// SIMATIC S7-200 project (STEP 7-Micro/WIN), CPU 224 CN REL 02.01

ORGANIZATION_BLOCK 主程序:OB1
TITLE=程序注释
BEGIN
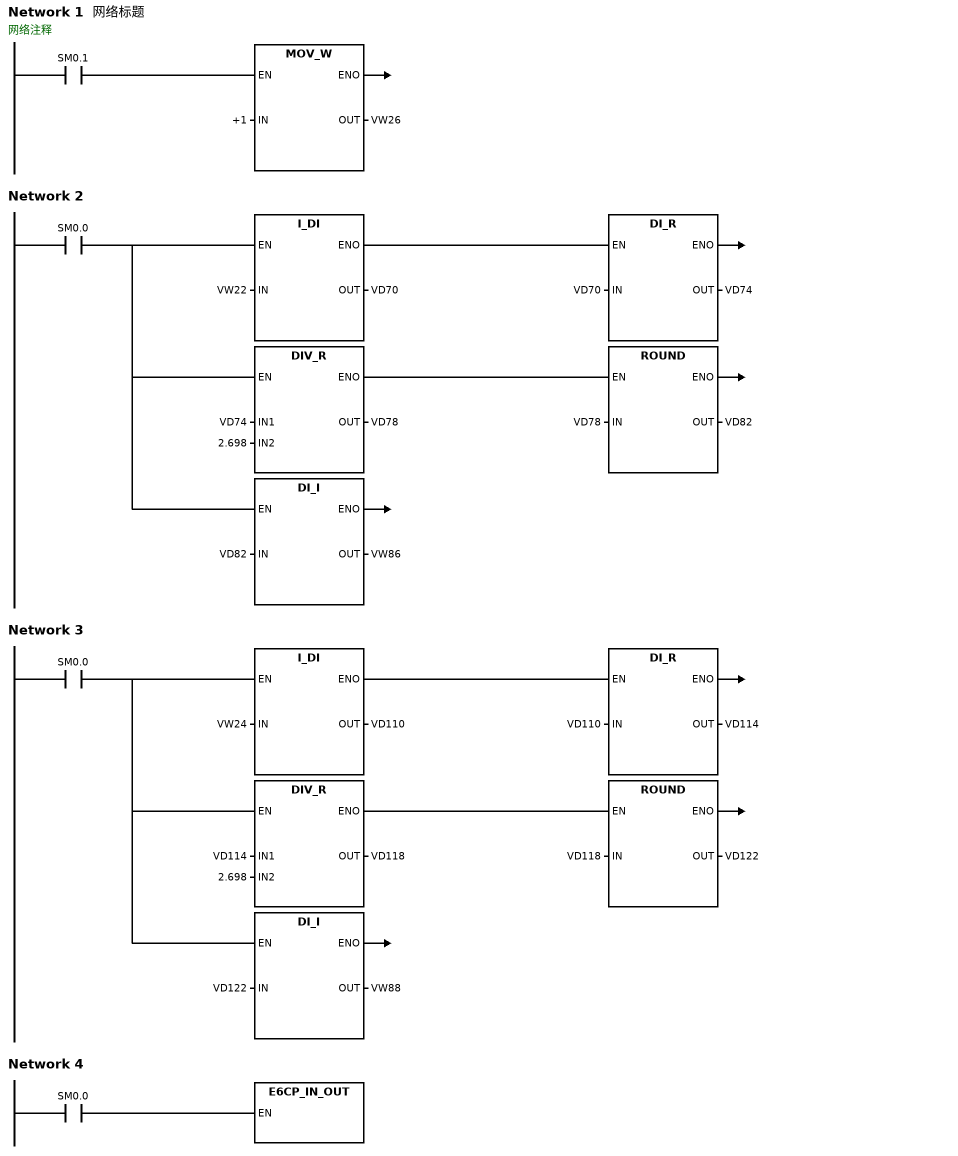
Network 1 // 网络标题
// 网络注释
LD     SM0.1
MOVW   +1, VW26
Network 2
LD     SM0.0
LPS
ITD    VW22, VD70
AENO
DTR    VD70, VD74
LRD
MOVR   VD74, VD78
AENO
/R     2.698, VD78
AENO
ROUND  VD78, VD82
LPP
DTI    VD82, VW86
Network 3
LD     SM0.0
LPS
ITD    VW24, VD110
AENO
DTR    VD110, VD114
LRD
MOVR   VD114, VD118
AENO
/R     2.698, VD118
AENO
ROUND  VD118, VD122
LPP
DTI    VD122, VW88
Network 4
LD     SM0.0
CALL   E6CP_IN_OUT:SBR4
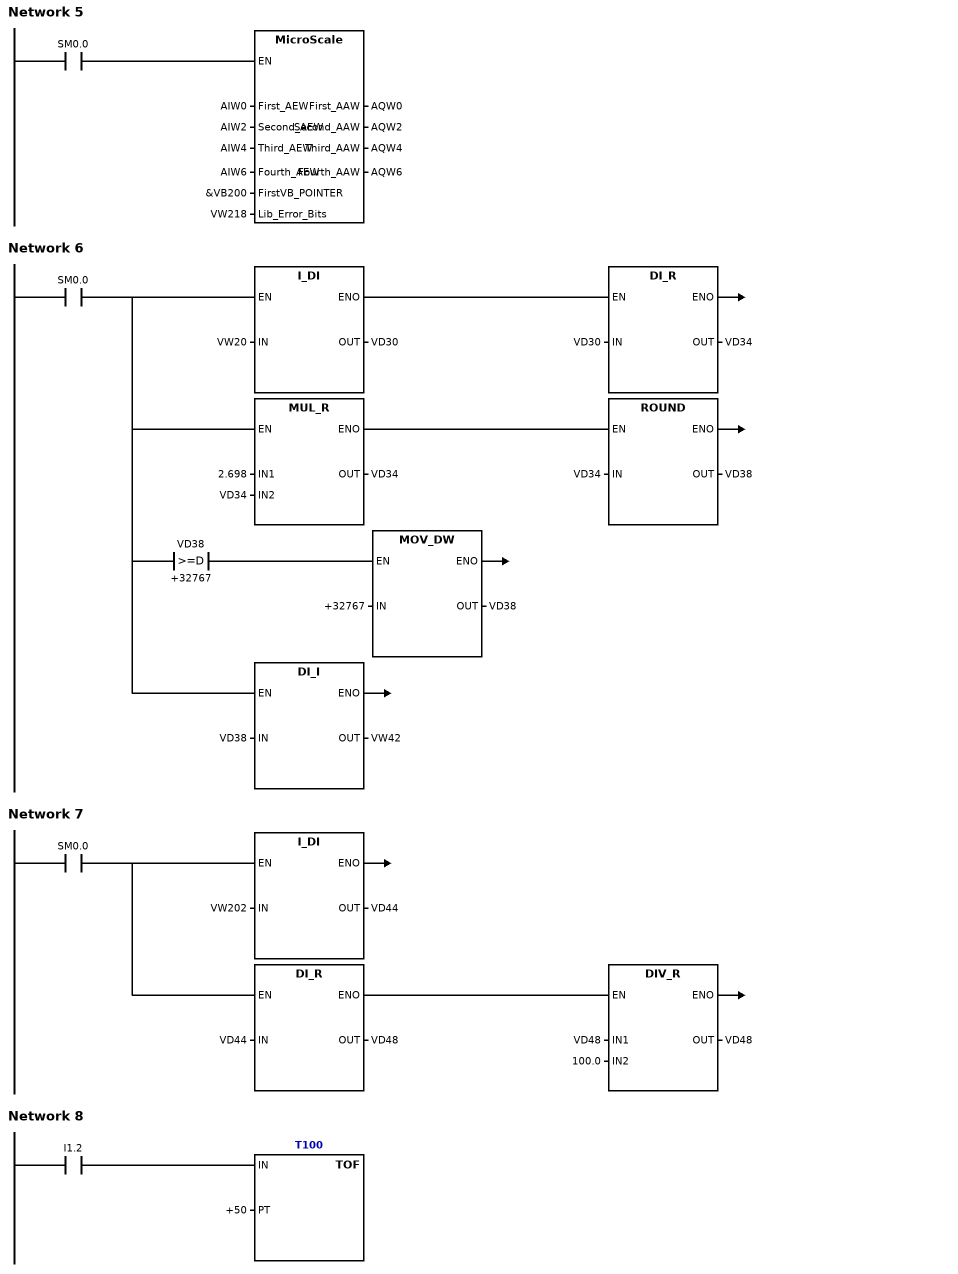
Network 5
LD     SM0.0
CALL   MicroScale:SBR3, AIW0, AIW2, AIW4, AIW6, &VB200, VW218, AQW0, AQW2, AQW4, AQW6
Network 6
LD     SM0.0
LPS
ITD    VW20, VD30
AENO
DTR    VD30, VD34
LRD
*R     2.698, VD34
AENO
ROUND  VD34, VD38
LRD
AD>=   VD38, +32767
MOVD   +32767, VD38
LPP
DTI    VD38, VW42
Network 7
LD     SM0.0
ITD    VW202, VD44
DTR    VD44, VD48
AENO
/R     100.0, VD48
Network 8
LD     I1.2
TOF    T100, +50
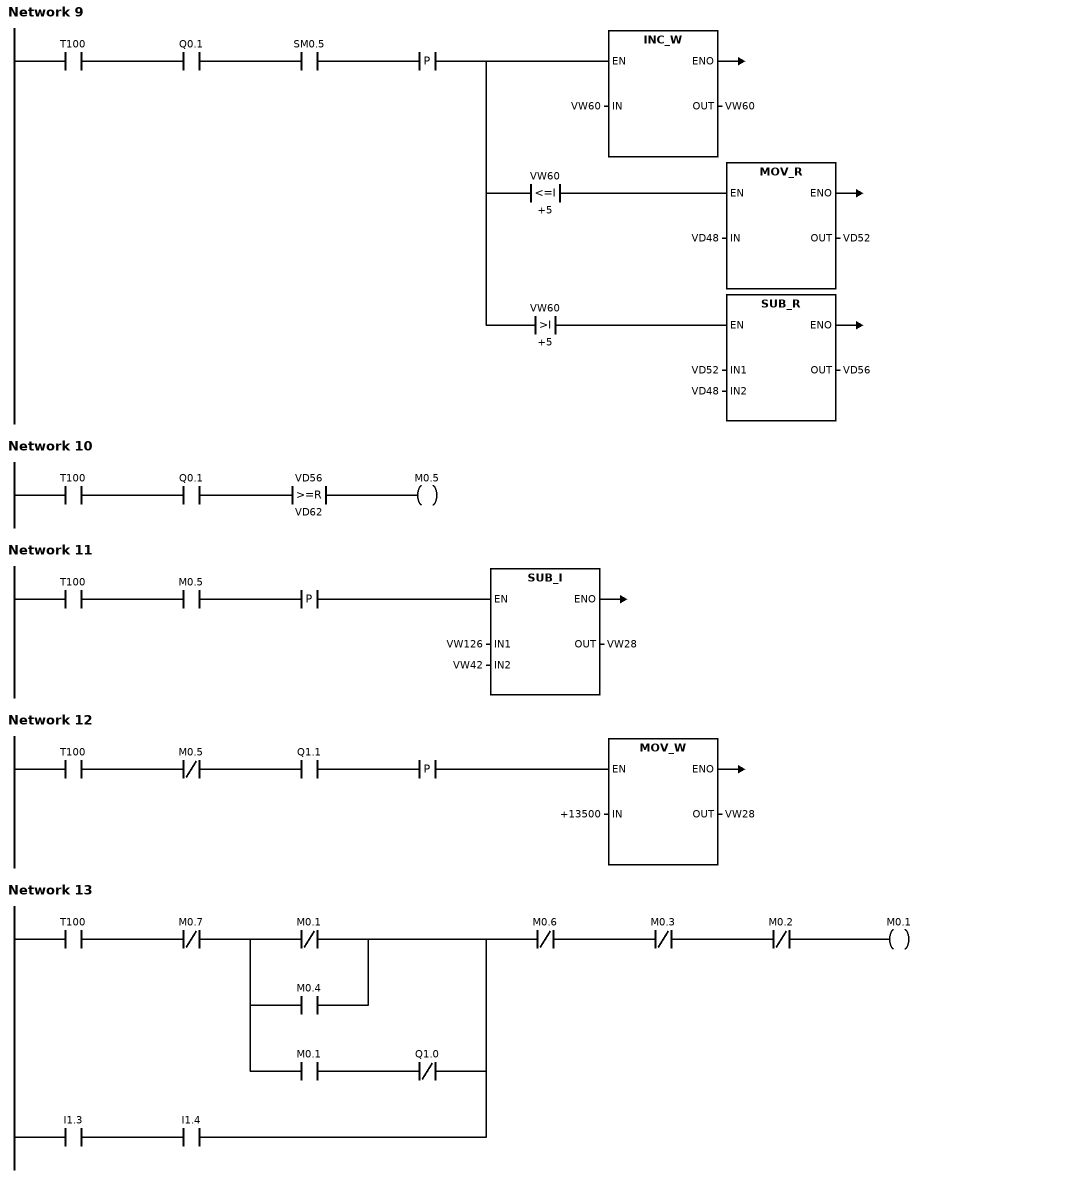
Network 9
LD     T100
A      Q0.1
A      SM0.5
EU
LPS
INCW   VW60
AW<=   VW60, +5
MOVR   VD48, VD52
LPP
AW>    VW60, +5
MOVR   VD52, VD56
-R     VD48, VD56
Network 10
LD     T100
A      Q0.1
AR>=   VD56, VD62
=      M0.5
Network 11
LD     T100
A      M0.5
EU
MOVW   VW126, VW28
-I     VW42, VW28
Network 12
LD     T100
AN     M0.5
A      Q1.1
EU
MOVW   +13500, VW28
Network 13
LD     T100
AN     M0.7
LDN    M0.1
O      M0.4
LD     M0.1
AN     Q1.0
OLD
ALD
LD     I1.3
A      I1.4
OLD
AN     M0.6
AN     M0.3
AN     M0.2
=      M0.1
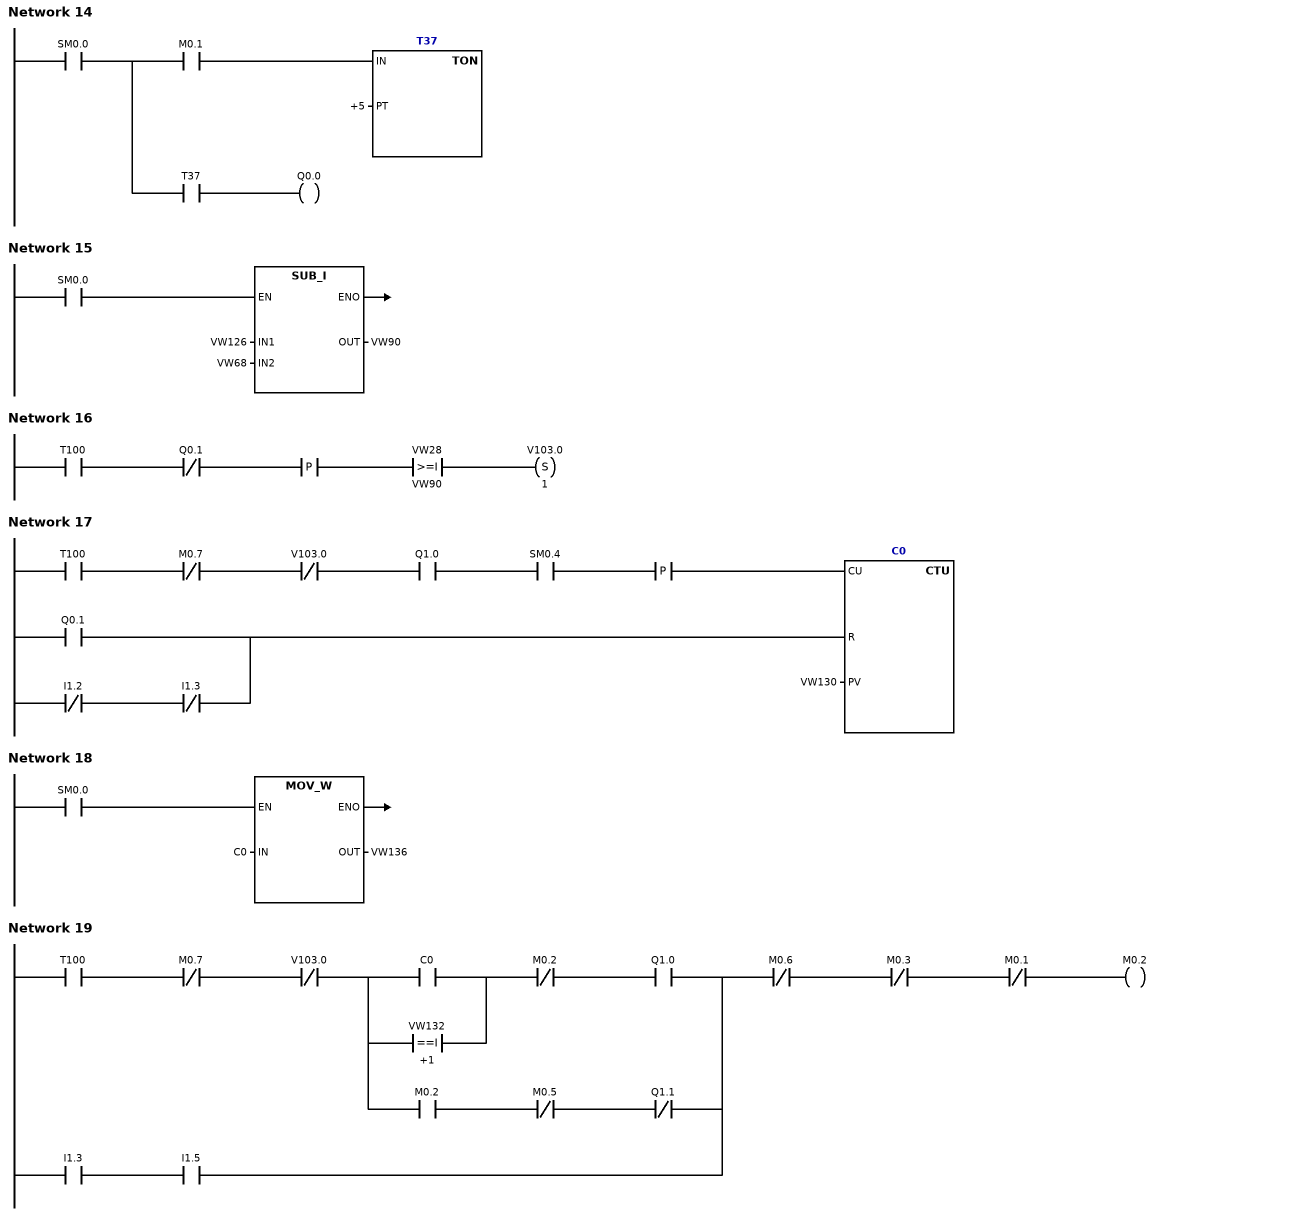
Network 14
LD     SM0.0
LPS
A      M0.1
TON    T37, +5
LPP
A      T37
=      Q0.0
Network 15
LD     SM0.0
MOVW   VW126, VW90
-I     VW68, VW90
Network 16
LD     T100
AN     Q0.1
EU
AW>=   VW28, VW90
S      V103.0, 1
Network 17
LD     T100
AN     M0.7
AN     V103.0
A      Q1.0
A      SM0.4
EU
LD     Q0.1
LDN    I1.2
AN     I1.3
OLD
CTU    C0, VW130
Network 18
LD     SM0.0
MOVW   C0, VW136
Network 19
LD     T100
AN     M0.7
AN     V103.0
LD     C0
OW=    VW132, +1
AN     M0.2
A      Q1.0
LD     M0.2
AN     M0.5
AN     Q1.1
OLD
ALD
LD     I1.3
A      I1.5
OLD
AN     M0.6
AN     M0.3
AN     M0.1
=      M0.2
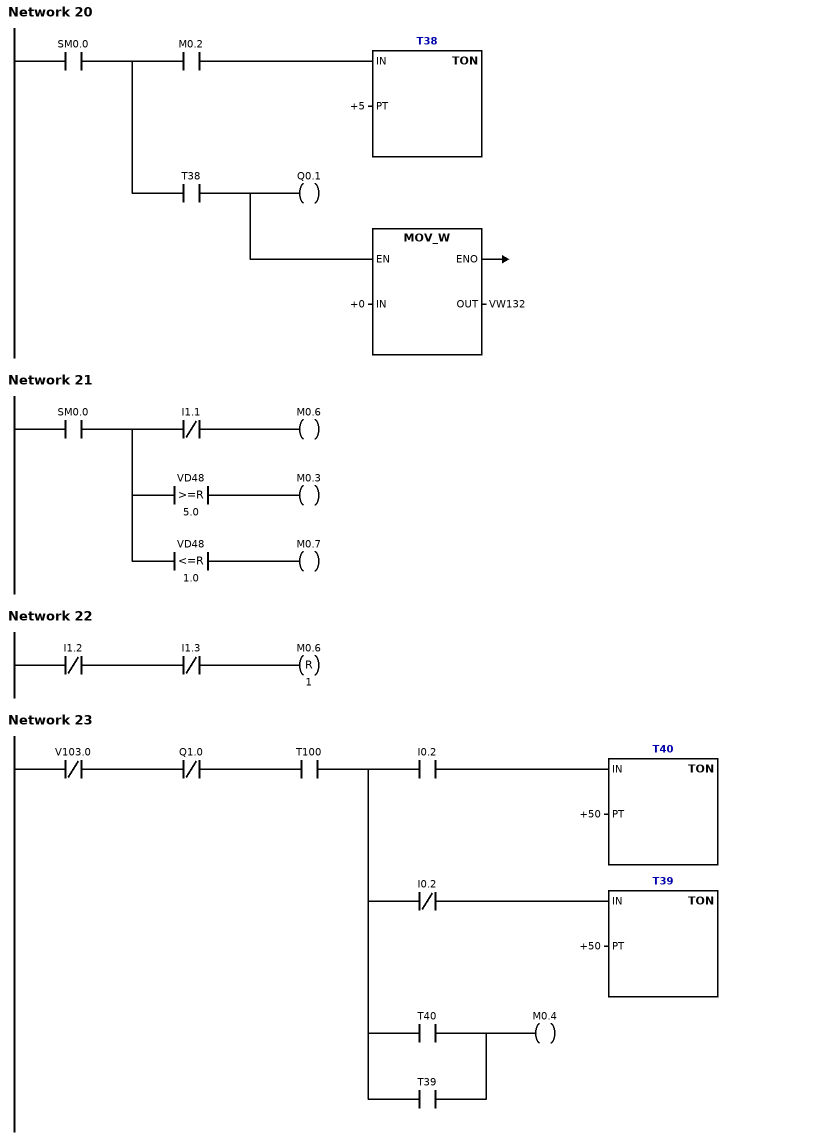
Network 20
LD     SM0.0
LPS
A      M0.2
TON    T38, +5
LPP
A      T38
=      Q0.1
MOVW   +0, VW132
Network 21
LD     SM0.0
LPS
AN     I1.1
=      M0.6
LRD
AR>=   VD48, 5.0
=      M0.3
LPP
AR<=   VD48, 1.0
=      M0.7
Network 22
LDN    I1.2
AN     I1.3
R      M0.6, 1
Network 23
LDN    V103.0
AN     Q1.0
A      T100
LPS
A      I0.2
TON    T40, +50
LRD
AN     I0.2
TON    T39, +50
LPP
LD     T40
O      T39
ALD
=      M0.4
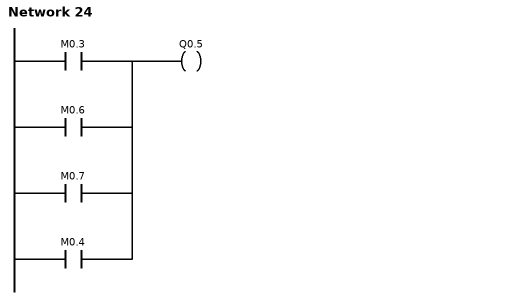
Network 24
LD     M0.3
O      M0.6
O      M0.7
O      M0.4
=      Q0.5
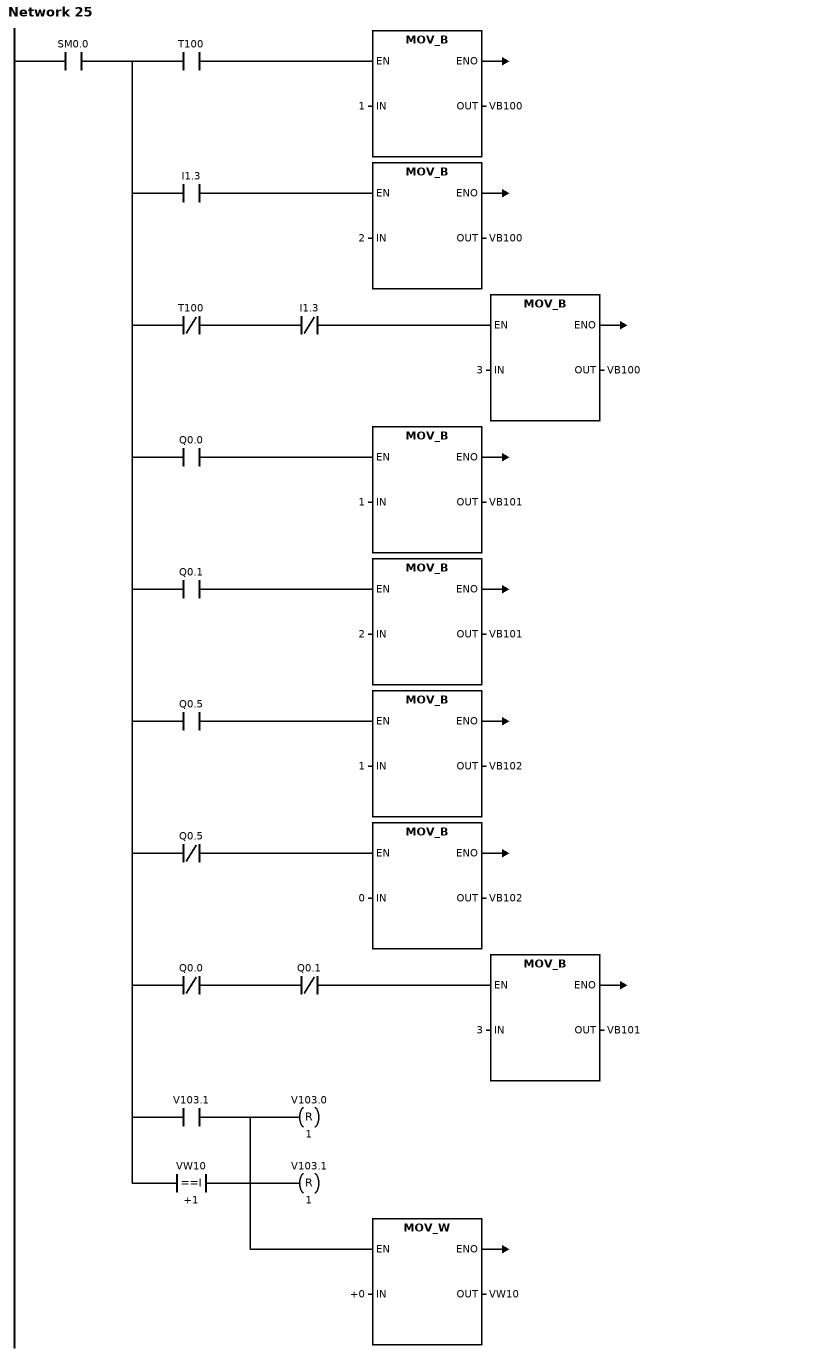
Network 25
LD     SM0.0
LPS
A      T100
MOVB   1, VB100
LRD
A      I1.3
MOVB   2, VB100
LRD
AN     T100
AN     I1.3
MOVB   3, VB100
LRD
A      Q0.0
MOVB   1, VB101
LRD
A      Q0.1
MOVB   2, VB101
LRD
A      Q0.5
MOVB   1, VB102
LRD
AN     Q0.5
MOVB   0, VB102
LRD
AN     Q0.0
AN     Q0.1
MOVB   3, VB101
LPP
LD     V103.1
OW=    VW10, +1
ALD
R      V103.0, 1
R      V103.1, 1
MOVW   +0, VW10
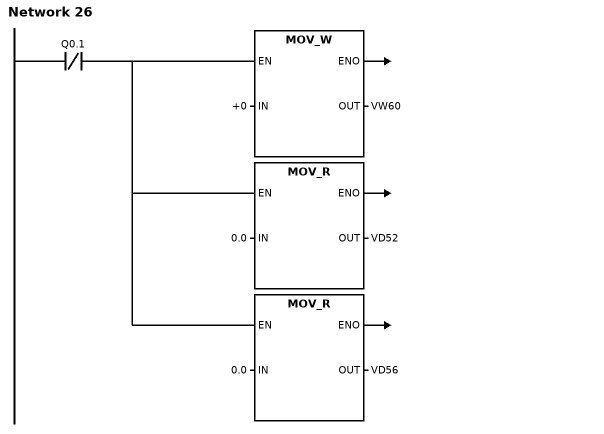
Network 26
LDN    Q0.1
MOVW   +0, VW60
MOVR   0.0, VD52
MOVR   0.0, VD56
END_ORGANIZATION_BLOCK

SUBROUTINE_BLOCK E6CP:SBR0
TITLE=子程序注释
VAR_INPUT
Input_Bit_7:BOOL;	// L0.0 
Input_Bit_6:BOOL;	// L0.1 
Input_Bit_5:BOOL;	// L0.2 
Input_Bit_4:BOOL;	// L0.3 
Input_Bit_3:BOOL;	// L0.4 
Input_Bit_2:BOOL;	// L0.5 
Input_Bit_1:BOOL;	// L0.6 
Input_Bit_0:BOOL;	// L0.7 
Input_Top:WORD;	// LW1 
Input_Bootom:WORD;	// LW3 
END_VAR
VAR_IN_OUT
Set_Zero:WORD;	// LW5 
END_VAR
VAR_OUTPUT
Output_Val:INT;	// LW7 
Top_Bit:BOOL;	// L9.0 
Bootom_Bit:BOOL;	// L9.1 
Out_Pulse:BOOL;	// L9.2 
END_VAR
BEGIN
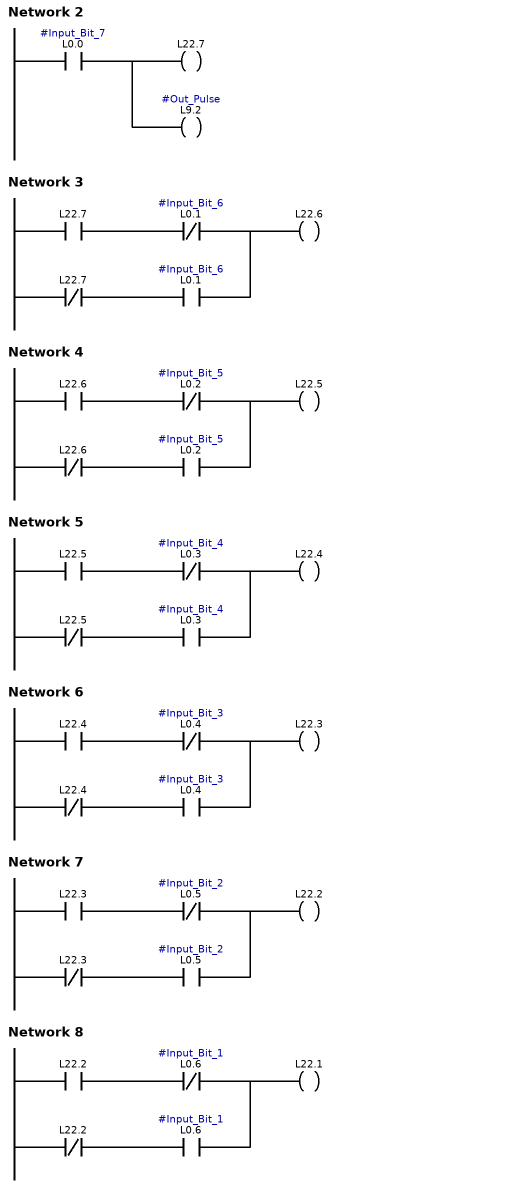
Network 2
LD     #Input_Bit_7:L0.0
=      L22.7
=      #Out_Pulse:L9.2
Network 3
LD     L22.7
AN     #Input_Bit_6:L0.1
LDN    L22.7
A      #Input_Bit_6:L0.1
OLD
=      L22.6
Network 4
LD     L22.6
AN     #Input_Bit_5:L0.2
LDN    L22.6
A      #Input_Bit_5:L0.2
OLD
=      L22.5
Network 5
LD     L22.5
AN     #Input_Bit_4:L0.3
LDN    L22.5
A      #Input_Bit_4:L0.3
OLD
=      L22.4
Network 6
LD     L22.4
AN     #Input_Bit_3:L0.4
LDN    L22.4
A      #Input_Bit_3:L0.4
OLD
=      L22.3
Network 7
LD     L22.3
AN     #Input_Bit_2:L0.5
LDN    L22.3
A      #Input_Bit_2:L0.5
OLD
=      L22.2
Network 8
LD     L22.2
AN     #Input_Bit_1:L0.6
LDN    L22.2
A      #Input_Bit_1:L0.6
OLD
=      L22.1
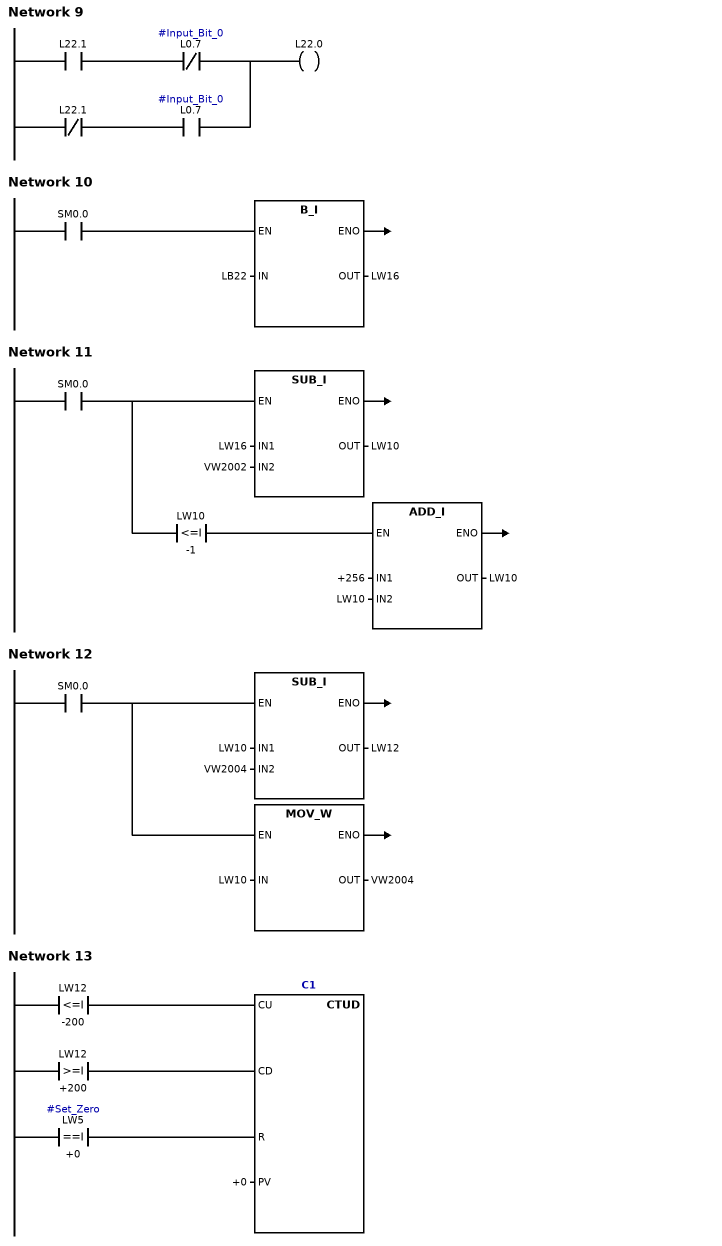
Network 9
LD     L22.1
AN     #Input_Bit_0:L0.7
LDN    L22.1
A      #Input_Bit_0:L0.7
OLD
=      L22.0
Network 10
LD     SM0.0
BTI    LB22, LW16
Network 11
LD     SM0.0
MOVW   LW16, LW10
-I     VW2002, LW10
AW<=   LW10, -1
+I     +256, LW10
Network 12
LD     SM0.0
MOVW   LW10, LW12
-I     VW2004, LW12
MOVW   LW10, VW2004
Network 13
LDW<=  LW12, -200
LDW>=  LW12, +200
LDW=   #Set_Zero:LW5, +0
CTUD   C1, +0
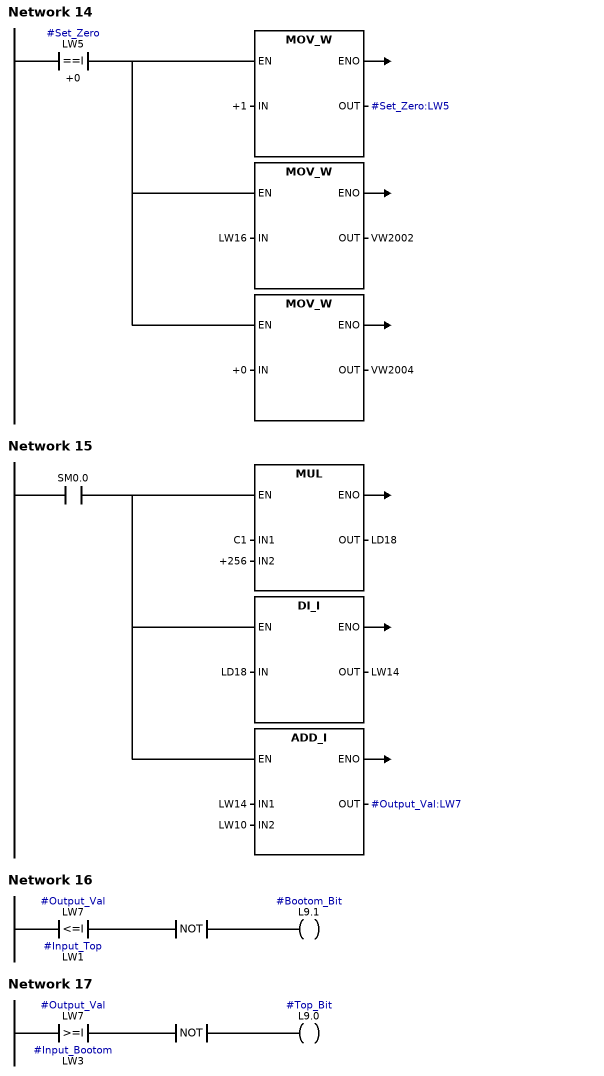
Network 14
LDW=   #Set_Zero:LW5, +0
MOVW   +1, #Set_Zero:LW5
MOVW   LW16, VW2002
MOVW   +0, VW2004
Network 15
LD     SM0.0
MOVW   C1, LW20
MUL    +256, LD18
DTI    LD18, LW14
MOVW   LW14, #Output_Val:LW7
+I     LW10, #Output_Val:LW7
Network 16
LDW<=  #Output_Val:LW7, #Input_Top:LW1
NOT
=      #Bootom_Bit:L9.1
Network 17
LDW>=  #Output_Val:LW7, #Input_Bootom:LW3
NOT
=      #Top_Bit:L9.0
END_SUBROUTINE_BLOCK

// SBR1: protected block, not included

// SBR2: protected block, not included

// SBR3: protected block, not included

SUBROUTINE_BLOCK E6CP_IN_OUT:SBR4
TITLE=
BEGIN
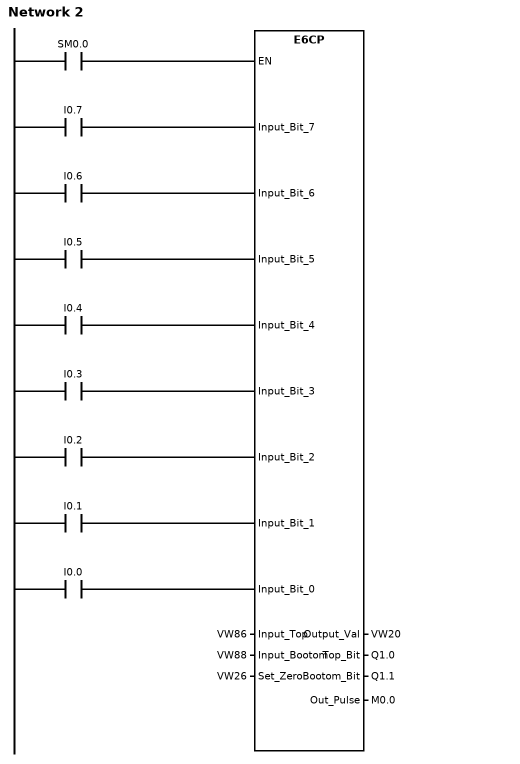
Network 2
LD     SM0.0
=      L60.0
LD     I0.7
=      L63.7
LD     I0.6
=      L63.6
LD     I0.5
=      L63.5
LD     I0.4
=      L63.4
LD     I0.3
=      L63.3
LD     I0.2
=      L63.2
LD     I0.1
=      L63.1
LD     I0.0
=      L63.0
LD     L60.0
CALL   E6CP:SBR0, L63.7, L63.6, L63.5, L63.4, L63.3, L63.2, L63.1, L63.0, VW86, VW88, VW26, VW20, Q1.0, Q1.1, M0.0
END_SUBROUTINE_BLOCK

DATA_BLOCK_TAB 用户定义1
BEGIN
VW22     +10000
VW24     0
VD62     1.0
VW68     8000
VW126    +12000
END_DATA_BLOCK_TAB

// (further data pages could not be read)
